FUNCTION_BLOCK EL3154
VAR
	_io : EL3xx4_Data;
	{attribute addProperty Name "WcState"}
	_wcState : WcStateInputToggle;
	{attribute addProperty Name "Info data"}
	_infoData : InfoDataAds;
END_VAR

PROPERTY IO : REFERENCE TO EL3xx4_Data
GET
IO REF= _io;
END_GET
END_PROPERTY

PROPERTY WcState : REFERENCE TO WcStateInputToggle
GET
WcState REF= _wcState;
END_GET
END_PROPERTY

END_FUNCTION_BLOCK

(* stored: Version 1.1.0.1, ProductVersion 3.1.4024.9
   POU EL3154: Id {18f8760f-82fc-07ae-04e5-e8f902630ac2}, SpecialFunc None
   Property IO: Id {909dbbc9-ace7-00ee-204d-0d19fdea600c}
   Get Get: Id {c144c5cc-720c-0cc6-08b1-22c155aa3fb6}
   Property WcState: Id {23e95868-0cb7-0c9c-1966-2306c08320d7}
   Get Get: Id {30ed9d74-5b6f-0cb2-07ee-617ba5e20c4a} *)
